PROGRAM Main
VAR
END_VAR

///Calling programs
PRG_Roughing();				
PRG_SampleChamber(); 		
//PRG_SDS();
//PRG_SPCA();
PRG_2_PMPS();
PRG_3_LOG();

END_PROGRAM

(* stored: Version 1.1.0.1, ProductVersion 3.1.4022.18
   POU Main: Id {ecf97ee3-9889-4850-9da7-1b720e899e44}, SpecialFunc None *)
